INTERFACE ITF_TopElement2_HMI_Connector_Command EXTENDS ITF_BaseTopElement_HMI_Connector_Command

END_INTERFACE

(* stored: Version 1.1.0.1
   Itf ITF_TopElement2_HMI_Connector_Command: Id {4dbc53df-24ff-0cc6-2eb5-680f3adcb6dc} *)
